Fanuc KAREL source: ks00045.KL

-- PROVISIONAL review KL for V770-1; original PC SHA256 8a6a02ceb244f5e2770d8840c3a3ad40a3ad4385c9e08b0eb6e2157377ff55fe
-- Incomplete behavior may be omitted. Consult companion uncertainty JSON. Do not deploy.
PROGRAM KS00045
%NOLOCKGROUP
BEGIN
  -- UNRESOLVED_PC offsets 5-13; opcodes 3F,75
  -- UNRESOLVED_PC offsets 18-27; opcodes 3F,75
  -- UNRESOLVED_PC offsets 32-46; opcodes 22,22,1E
  -- UNRESOLVED_PC offsets 51-55; opcodes 7F
END KS00045
